PROGRAM MAIN
VAR
END_VAR

END_PROGRAM

(* stored: Version 1.1.0.1
   POU MAIN: Id {75ffc185-3e69-4fa4-b952-72ead9b4295f} *)
